// TIA Portal V20 export
TYPE "ItemDir"
// stored: Access Published, Namespace LineA1
   STRUCT
      Straight : Bool;
      toRight : Bool;
      toLeft : Bool;
   END_STRUCT;
END_TYPE
